LIN {X 0,Y 60.716,Z 312.384,A -85,B 0,C 180,E1 -29461.22,E2 -29461.22} C_VEL
LIN {X 0,Y 58.046,Z 307.358,A -85,B 0,C 180,E1 -29469.715,E2 -29469.715} C_VEL
LIN {X 0,Y 56.371,Z 305.582,A -85,B 0,C 180,E1 -29475.475,E2 -29475.475} C_VEL
LIN {X 0,Y 55.559,Z 303.266,A -85,B 0,C 180,E1 -29480.778,E2 -29480.778} C_VEL
LIN {X 0,Y 54.306,Z 302.152,A -85,B 0,C 180,E1 -29488.836,E2 -29488.836} C_VEL
LIN {X 0,Y 53.915,Z 301.998,A -85,B 0,C 180,E1 -29493.79,E2 -29493.79} C_VEL
LIN {X 0,Y 53.664,Z 302.515,A -85,B 0,C 180,E1 -29497.928,E2 -29497.928} C_VEL
LIN {X 0,Y 53.314,Z 303.941,A -85,B 0,C 180,E1 -29501.896,E2 -29501.896} C_VEL
LIN {X 0,Y 53.027,Z 308.841,A -85,B 0,C 180,E1 -29512.371,E2 -29512.371} C_VEL
LIN {X 0,Y 53.437,Z 309.628,A -85,B 0,C 180,E1 -29515.134,E2 -29515.134} C_VEL
LIN {X 0,Y 54.909,Z 313.062,A -85,B 0,C 180,E1 -29523.678,E2 -29523.678} C_VEL
LIN {X 0,Y 56.343,Z 316.547,A -85,B 0,C 180,E1 -29529.884,E2 -29529.884} C_VEL
LIN {X 0,Y 58.459,Z 322.301,A -85,B 0,C 180,E1 -29537.951,E2 -29537.951} C_VEL
LIN {X 0,Y 60.242,Z 328.035,A -85,B 0,C 180,E1 -29544.566,E2 -29544.566} C_VEL
LIN {X 0,Y 60.742,Z 331.305,A -85,B 0,C 180,E1 -29547.577,E2 -29547.577} C_VEL
LIN {X 0,Y 60.313,Z 334.364,A -85,B 0,C 180,E1 -29549.694,E2 -29549.694} C_VEL
LIN {X 0,Y 57.768,Z 345.368,A -85,B 0,C 180,E1 -29557.476,E2 -29557.476} C_VEL
LIN {X 0,Y 56.308,Z 350.331,A -85,B 0,C 180,E1 -29561.507,E2 -29561.507} C_VEL
LIN {X 0,Y 50.983,Z 359.168,A -85,B 0,C 180,E1 -29569.096,E2 -29569.096} C_VEL
LIN {X 0,Y 45.942,Z 367.817,A -85,B 0,C 180,E1 -29580.186,E2 -29580.186} C_VEL
LIN {X 0,Y 42.807,Z 374.789,A -85,B 0,C 180,E1 -29593.302,E2 -29593.302} C_VEL
LIN {X 0,Y 41.908,Z 379.494,A -85,B 0,C 180,E1 -29605.189,E2 -29605.189} C_VEL
LIN {X 0,Y 42.054,Z 382.623,A -85,B 0,C 180,E1 -29614.792,E2 -29614.792} C_VEL
LIN {X 0,Y 43.107,Z 386.22,A -85,B 0,C 180,E1 -29629.029,E2 -29629.029} C_VEL
LIN {X 0,Y 45.194,Z 388.132,A -85,B 0,C 180,E1 -29637.807,E2 -29637.807} C_VEL
LIN {X 0,Y 51.933,Z 390.826,A -85,B 0,C 180,E1 -29652.58,E2 -29652.58} C_VEL
LIN {X 0,Y 61.527,Z 392.195,A -85,B 0,C 180,E1 -29663.088,E2 -29663.088} C_VEL
LIN {X 0,Y 72.679,Z 392.248,A -85,B 0,C 180,E1 -29670.489,E2 -29670.489} C_VEL
LIN {X 0,Y 84.73,Z 390.994,A -85,B 0,C 180,E1 -29675.836,E2 -29675.836} C_VEL
LIN {X 0,Y 91.024,Z 389.845,A -85,B 0,C 180,E1 -29677.895,E2 -29677.895} C_VEL
LIN {X 0,Y 93.755,Z 389.205,A -85,B 0,C 180,E1 -29679.343,E2 -29679.343} C_VEL
LIN {X 0,Y 80.434,Z 391.186,A -85,B 0,C 180,E1 -29683.967,E2 -29683.967} C_VEL
LIN {X 0,Y 70.96,Z 391.617,A -85,B 0,C 180,E1 -29688.568,E2 -29688.568} C_VEL
LIN {X 0,Y 63.384,Z 391.312,A -85,B 0,C 180,E1 -29693.626,E2 -29693.626} C_VEL
LIN {X 0,Y 56.222,Z 390.333,A -85,B 0,C 180,E1 -29700.253,E2 -29700.253} C_VEL
LIN {X 0,Y 47.716,Z 387.672,A -85,B 0,C 180,E1 -29713.041,E2 -29713.041} C_VEL
LIN {X 0,Y 42.291,Z 383.509,A -85,B 0,C 180,E1 -29729.89,E2 -29729.89} C_VEL
LIN {X 0,Y 40.912,Z 378.594,A -85,B 0,C 180,E1 -29746.6,E2 -29746.6} C_VEL
LIN {X 0,Y 42.587,Z 372.224,A -85,B 0,C 180,E1 -29763.016,E2 -29763.016} C_VEL
LIN {X 0,Y 46.467,Z 364.513,A -85,B 0,C 180,E1 -29776.889,E2 -29776.889} C_VEL
LIN {X 0,Y 51.445,Z 356.174,A -85,B 0,C 180,E1 -29787.065,E2 -29787.065} C_VEL
LIN {X 0,Y 56.882,Z 347.135,A -85,B 0,C 180,E1 -29794.55,E2 -29794.55} C_VEL
LIN {X 0,Y 59.718,Z 342.179,A -85,B 0,C 180,E1 -29797.602,E2 -29797.602} C_VEL
LIN {X 0,Y 61.132,Z 334.574,A -85,B 0,C 180,E1 -29803.294,E2 -29803.294} C_VEL
LIN {X 0,Y 61.35,Z 332.923,A -85,B 0,C 180,E1 -29804.489,E2 -29804.489} C_VEL
LIN {X 0,Y 60.3,Z 328.115,A -85,B 0,C 180,E1 -29809.376,E2 -29809.376} C_VEL
LIN {X 0,Y 59.125,Z 324.115,A -85,B 0,C 180,E1 -29813.986,E2 -29813.986} C_VEL
LIN {X 0,Y 56.439,Z 317.616,A -85,B 0,C 180,E1 -29823.356,E2 -29823.356} C_VEL
LIN {X 0,Y 54.803,Z 314.262,A -85,B 0,C 180,E1 -29829.882,E2 -29829.882} C_VEL
LIN {X 0,Y 52.508,Z 309.531,A -85,B 0,C 180,E1 -29843.426,E2 -29843.426} C_VEL
LIN {X 0,Y 51.489,Z 308.683,A -85,B 0,C 180,E1 -29854.149,E2 -29854.149} C_VEL
LIN {X 0,Y 51.797,Z 308.515,A -85,B 0,C 180,E1 -29864.264,E2 -29864.264} C_VEL
LIN {X 0,Y 52.94,Z 309.058,A -85,B 0,C 180,E1 -29872.38,E2 -29872.38} C_VEL
LIN {X 0,Y 53.437,Z 309.628,A -85,B 0,C 180,E1 -29875.134,E2 -29875.134} C_VEL
LIN {X 0,Y 54.073,Z 310.974,A -85,B 0,C 180,E1 -29878.941,E2 -29878.941} C_VEL
LIN {X 0,Y 54.486,Z 314.348,A -85,B 0,C 180,E1 -29884.001,E2 -29884.001} C_VEL
LIN {X 0,Y 54.414,Z 318.577,A -85,B 0,C 180,E1 -29888.441,E2 -29888.441} C_VEL
LIN {X 0,Y 54.152,Z 327.952,A -85,B 0,C 180,E1 -29897.401,E2 -29897.401} C_VEL
LIN {X 0,Y 54.569,Z 330.721,A -85,B 0,C 180,E1 -29900.693,E2 -29900.693} C_VEL
LIN {X 0,Y 54.973,Z 334.381,A -85,B 0,C 180,E1 -29904.759,E2 -29904.759} C_VEL
LIN {X 0,Y 52.046,Z 344.757,A -85,B 0,C 180,E1 -29912.704,E2 -29912.704} C_VEL
LIN {X 0,Y 50.55,Z 349.485,A -85,B 0,C 180,E1 -29916.925,E2 -29916.925} C_VEL
LIN {X 0,Y 44.772,Z 358.482,A -85,B 0,C 180,E1 -29925.058,E2 -29925.058} C_VEL
LIN {X 0,Y 39.175,Z 367.209,A -85,B 0,C 180,E1 -29937.437,E2 -29937.437} C_VEL
LIN {X 0,Y 35.705,Z 374.24,A -85,B 0,C 180,E1 -29952.826,E2 -29952.826} C_VEL
LIN {X 0,Y 34.905,Z 379.848,A -85,B 0,C 180,E1 -29969.998,E2 -29969.998} C_VEL
LIN {X 0,Y 35.339,Z 382.791,A -85,B 0,C 180,E1 -29981.469,E2 -29981.469} C_VEL
LIN {X 0,Y 39.079,Z 387.199,A -85,B 0,C 180,E1 -30002.648,E2 -30002.648} C_VEL
LIN {X 0,Y 46.959,Z 390.173,A -85,B 0,C 180,E1 -30018.441,E2 -30018.441} C_VEL
LIN {X 0,Y 57.536,Z 391.813,A -85,B 0,C 180,E1 -30028.76,E2 -30028.76} C_VEL
LIN {X 0,Y 69.448,Z 392.107,A -85,B 0,C 180,E1 -30035.61,E2 -30035.61} C_VEL
LIN {X 0,Y 75.681,Z 391.763,A -85,B 0,C 180,E1 -30038.218,E2 -30038.218} C_VEL
LIN {X 0,Y 76.461,Z 391.653,A -85,B 0,C 180,E1 -30039.648,E2 -30039.648} C_VEL
LIN {X 0,Y 65.683,Z 391.772,A -85,B 0,C 180,E1 -30044.355,E2 -30044.355} C_VEL
LIN {X 0,Y 53.748,Z 390.589,A -85,B 0,C 180,E1 -30052.478,E2 -30052.478} C_VEL
LIN {X 0,Y 46.797,Z 389.001,A -85,B 0,C 180,E1 -30059.99,E2 -30059.99} C_VEL
LIN {X 0,Y 38.984,Z 385.698,A -85,B 0,C 180,E1 -30074.48,E2 -30074.48} C_VEL
LIN {X 0,Y 34.398,Z 380.739,A -85,B 0,C 180,E1 -30095.193,E2 -30095.193} C_VEL
LIN {X 0,Y 34.3,Z 375.093,A -85,B 0,C 180,E1 -30115.018,E2 -30115.018} C_VEL
LIN {X 0,Y 37.056,Z 368.741,A -85,B 0,C 180,E1 -30131.453,E2 -30131.453} C_VEL
LIN {X 0,Y 42.273,Z 360.323,A -85,B 0,C 180,E1 -30145.798,E2 -30145.798} C_VEL
LIN {X 0,Y 48.602,Z 350.774,A -85,B 0,C 180,E1 -30155.913,E2 -30155.913} C_VEL
LIN {X 0,Y 53.498,Z 343.032,A -85,B 0,C 180,E1 -30161.366,E2 -30161.366} C_VEL
LIN {X 0,Y 54.525,Z 339.734,A -85,B 0,C 180,E1 -30163.986,E2 -30163.986} C_VEL
LIN {X 0,Y 55.408,Z 334.818,A -85,B 0,C 180,E1 -30168.185,E2 -30168.185} C_VEL
LIN {X 0,Y 54.271,Z 329.443,A -85,B 0,C 180,E1 -30174.997,E2 -30174.997} C_VEL
LIN {X 0,Y 52.71,Z 324.789,A -85,B 0,C 180,E1 -30182.232,E2 -30182.232} C_VEL
LIN {X 0,Y 52.023,Z 322.703,A -85,B 0,C 180,E1 -30185.865,E2 -30185.865} C_VEL
LIN {X 0,Y 50.614,Z 319.24,A -85,B 0,C 180,E1 -30193.97,E2 -30193.97} C_VEL
LIN {X 0,Y 49.38,Z 315.79,A -85,B 0,C 180,E1 -30205.311,E2 -30205.311} C_VEL
LIN {X 0,Y 48.742,Z 315.216,A -85,B 0,C 180,E1 -30214.381,E2 -30214.381} C_VEL
LIN {X 0,Y 48.976,Z 315.067,A -85,B 0,C 180,E1 -30223.332,E2 -30223.332} C_VEL
LIN {X 0,Y 50.04,Z 315.547,A -85,B 0,C 180,E1 -30231.936,E2 -30231.936} C_VEL
LIN {X 0,Y 50.494,Z 316.572,A -85,B 0,C 180,E1 -30235.72,E2 -30235.72} C_VEL
LIN {X 0,Y 51.517,Z 319.997,A -85,B 0,C 180,E1 -30243.92,E2 -30243.92} C_VEL
LIN {X 0,Y 52.824,Z 324.176,A -85,B 0,C 180,E1 -30251.521,E2 -30251.521} C_VEL
LIN {X 0,Y 54.208,Z 329.381,A -85,B 0,C 180,E1 -30258.922,E2 -30258.922} C_VEL
LIN {X 0,Y 54.569,Z 330.721,A -85,B 0,C 180,E1 -30260.693,E2 -30260.693} C_VEL
LIN {X 0,Y 54.558,Z 332.559,A -85,B 0,C 180,E1 -30262.483,E2 -30262.483} C_VEL
LIN {X 0,Y 53.326,Z 335.803,A -85,B 0,C 180,E1 -30264.371,E2 -30264.371} C_VEL
LIN {X 0,Y 51.274,Z 339.05,A -85,B 0,C 180,E1 -30265.645,E2 -30265.645} C_VEL
LIN {X 0,Y 47.111,Z 344.69,A -85,B 0,C 180,E1 -30267.889,E2 -30267.889} C_VEL
LIN {X 0,Y 45.301,Z 347.952,A -85,B 0,C 180,E1 -30270.404,E2 -30270.404} C_VEL
LIN {X 0,Y 43.976,Z 350.677,A -85,B 0,C 180,E1 -30272.962,E2 -30272.962} C_VEL
LIN {X 0,Y 37.684,Z 359.374,A -85,B 0,C 180,E1 -30281.754,E2 -30281.754} C_VEL
LIN {X 0,Y 31.666,Z 367.857,A -85,B 0,C 180,E1 -30296.297,E2 -30296.297} C_VEL
LIN {X 0,Y 28.279,Z 374.686,A -85,B 0,C 180,E1 -30315.608,E2 -30315.608} C_VEL
LIN {X 0,Y 28.17,Z 380.088,A -85,B 0,C 180,E1 -30337.164,E2 -30337.164} C_VEL
LIN {X 0,Y 31.613,Z 385.2,A -85,B 0,C 180,E1 -30363.762,E2 -30363.762} C_VEL
LIN {X 0,Y 37.538,Z 388.017,A -85,B 0,C 180,E1 -30378.491,E2 -30378.491} C_VEL
LIN {X 0,Y 48.259,Z 390.554,A -85,B 0,C 180,E1 -30390.897,E2 -30390.897} C_VEL
LIN {X 0,Y 60.433,Z 391.783,A -85,B 0,C 180,E1 -30398.485,E2 -30398.485} C_VEL
LIN {X 0,Y 60.519,Z 391.753,A -85,B 0,C 180,E1 -30399.603,E2 -30399.603} C_VEL
LIN {X 0,Y 50.89,Z 390.609,A -85,B 0,C 180,E1 -30405.168,E2 -30405.168} C_VEL
LIN {X 0,Y 42.516,Z 388.752,A -85,B 0,C 180,E1 -30412.648,E2 -30412.648} C_VEL
LIN {X 0,Y 33.366,Z 385.23,A -85,B 0,C 180,E1 -30427.617,E2 -30427.617} C_VEL
LIN {X 0,Y 27.735,Z 380.268,A -85,B 0,C 180,E1 -30450.431,E2 -30450.431} C_VEL
LIN {X 0,Y 27.244,Z 374.435,A -85,B 0,C 180,E1 -30475.377,E2 -30475.377} C_VEL
LIN {X 0,Y 30.793,Z 367.38,A -85,B 0,C 180,E1 -30496.809,E2 -30496.809} C_VEL
LIN {X 0,Y 35.668,Z 360.447,A -85,B 0,C 180,E1 -30510.002,E2 -30510.002} C_VEL
LIN {X 0,Y 41.664,Z 352.31,A -85,B 0,C 180,E1 -30519.712,E2 -30519.712} C_VEL
LIN {X 0,Y 48.311,Z 342.597,A -85,B 0,C 180,E1 -30526.916,E2 -30526.916} C_VEL
LIN {X 0,Y 49.59,Z 337.634,A -85,B 0,C 180,E1 -30531.654,E2 -30531.654} C_VEL
LIN {X 0,Y 48.943,Z 333.355,A -85,B 0,C 180,E1 -30537.942,E2 -30537.942} C_VEL
LIN {X 0,Y 47.869,Z 328.994,A -85,B 0,C 180,E1 -30545.964,E2 -30545.964} C_VEL
LIN {X 0,Y 46.91,Z 325.511,A -85,B 0,C 180,E1 -30554.351,E2 -30554.351} C_VEL
LIN {X 0,Y 46.141,Z 323.114,A -85,B 0,C 180,E1 -30562.477,E2 -30562.477} C_VEL
LIN {X 0,Y 45.657,Z 321.682,A -85,B 0,C 180,E1 -30572.509,E2 -30572.509} C_VEL
LIN {X 0,Y 45.787,Z 321.464,A -85,B 0,C 180,E1 -30582.133,E2 -30582.133} C_VEL
LIN {X 0,Y 46.731,Z 321.903,A -85,B 0,C 180,E1 -30591.361,E2 -30591.361} C_VEL
LIN {X 0,Y 47.022,Z 323.048,A -85,B 0,C 180,E1 -30595.404,E2 -30595.404} C_VEL
LIN {X 0,Y 47.743,Z 326.68,A -85,B 0,C 180,E1 -30604.231,E2 -30604.231} C_VEL
LIN {X 0,Y 48.495,Z 330.562,A -85,B 0,C 180,E1 -30611.504,E2 -30611.504} C_VEL
LIN {X 0,Y 49.287,Z 335.135,A -85,B 0,C 180,E1 -30618.591,E2 -30618.591} C_VEL
LIN {X 0,Y 49.339,Z 336.759,A -85,B 0,C 180,E1 -30620.603,E2 -30620.603} C_VEL
LIN {X 0,Y 45.669,Z 346.976,A -85,B 0,C 180,E1 -30629.433,E2 -30629.433} C_VEL
LIN {X 0,Y 45.301,Z 347.952,A -85,B 0,C 180,E1 -30630.404,E2 -30630.404} C_VEL
LIN {X 0,Y 43.757,Z 350.87,A -85,B 0,C 180,E1 -30633.014,E2 -30633.014} C_VEL
LIN {X 0,Y 41.514,Z 353.649,A -85,B 0,C 180,E1 -30635.127,E2 -30635.127} C_VEL
LIN {X 0,Y 38.792,Z 356.232,A -85,B 0,C 180,E1 -30636.972,E2 -30636.972} C_VEL
LIN {X 0,Y 28.057,Z 364.422,A -85,B 0,C 180,E1 -30645.277,E2 -30645.277} C_VEL
LIN {X 0,Y 24.543,Z 367.912,A -85,B 0,C 180,E1 -30653.085,E2 -30653.085} C_VEL
LIN {X 0,Y 20.966,Z 375.052,A -85,B 0,C 180,E1 -30680.349,E2 -30680.349} C_VEL
LIN {X 0,Y 21.261,Z 378.672,A -85,B 0,C 180,E1 -30699.51,E2 -30699.51} C_VEL
LIN {X 0,Y 22.751,Z 381.611,A -85,B 0,C 180,E1 -30717.601,E2 -30717.601} C_VEL
LIN {X 0,Y 28.253,Z 385.172,A -85,B 0,C 180,E1 -30738.262,E2 -30738.262} C_VEL
LIN {X 0,Y 39.035,Z 388.662,A -85,B 0,C 180,E1 -30754.179,E2 -30754.179} C_VEL
LIN {X 0,Y 45.234,Z 389.927,A -85,B 0,C 180,E1 -30758.776,E2 -30758.776} C_VEL
LIN {X 0,Y 45.057,Z 389.877,A -85,B 0,C 180,E1 -30759.364,E2 -30759.364} C_VEL
LIN {X 0,Y 34.775,Z 387.17,A -85,B 0,C 180,E1 -30768.326,E2 -30768.326} C_VEL
LIN {X 0,Y 24.541,Z 382.499,A -85,B 0,C 180,E1 -30787.983,E2 -30787.983} C_VEL
LIN {X 0,Y 20.01,Z 377.129,A -85,B 0,C 180,E1 -30817.832,E2 -30817.832} C_VEL
LIN {X 0,Y 21.004,Z 371.715,A -85,B 0,C 180,E1 -30845.323,E2 -30845.323} C_VEL
LIN {X 0,Y 25.297,Z 365.423,A -85,B 0,C 180,E1 -30866.02,E2 -30866.02} C_VEL
LIN {X 0,Y 31.266,Z 358.122,A -85,B 0,C 180,E1 -30879.707,E2 -30879.707} C_VEL
LIN {X 0,Y 39.257,Z 348.201,A -85,B 0,C 180,E1 -30889.726,E2 -30889.726} C_VEL
LIN {X 0,Y 43.096,Z 342.821,A -85,B 0,C 180,E1 -30893.252,E2 -30893.252} C_VEL
LIN {X 0,Y 43.721,Z 341.086,A -85,B 0,C 180,E1 -30895.02,E2 -30895.02} C_VEL
LIN {X 0,Y 43.82,Z 338.697,A -85,B 0,C 180,E1 -30898.762,E2 -30898.762} C_VEL
LIN {X 0,Y 43.376,Z 335.116,A -85,B 0,C 180,E1 -30905.911,E2 -30905.911} C_VEL
LIN {X 0,Y 43.101,Z 333.047,A -85,B 0,C 180,E1 -30910.711,E2 -30910.711} C_VEL
LIN {X 0,Y 42.589,Z 330.414,A -85,B 0,C 180,E1 -30918.71,E2 -30918.71} C_VEL
LIN {X 0,Y 42.234,Z 328.761,A -85,B 0,C 180,E1 -30926.309,E2 -30926.309} C_VEL
LIN {X 0,Y 42.137,Z 328.272,A -85,B 0,C 180,E1 -30929.989,E2 -30929.989} C_VEL
LIN {X 0,Y 42.261,Z 327.696,A -85,B 0,C 180,E1 -30940.585,E2 -30940.585} C_VEL
LIN {X 0,Y 43.067,Z 328.096,A -85,B 0,C 180,E1 -30950.619,E2 -30950.619} C_VEL
LIN {X 0,Y 43.323,Z 331.287,A -85,B 0,C 180,E1 -30960.011,E2 -30960.011} C_VEL
LIN {X 0,Y 43.54,Z 334.374,A -85,B 0,C 180,E1 -30966.964,E2 -30966.964} C_VEL
LIN {X 0,Y 43.802,Z 339.224,A -85,B 0,C 180,E1 -30975.697,E2 -30975.697} C_VEL
LIN {X 0,Y 39.58,Z 348.685,A -85,B 0,C 180,E1 -30984.752,E2 -30984.752} C_VEL
LIN {X 0,Y 39.077,Z 349.777,A -85,B 0,C 180,E1 -30985.939,E2 -30985.939} C_VEL
LIN {X 0,Y 32.076,Z 358.552,A -85,B 0,C 180,E1 -30994.749,E2 -30994.749} C_VEL
LIN {X 0,Y 25.114,Z 367.127,A -85,B 0,C 180,E1 -31010.973,E2 -31010.973} C_VEL
LIN {X 0,Y 24.543,Z 367.912,A -85,B 0,C 180,E1 -31013.085,E2 -31013.085} C_VEL
LIN {X 0,Y 21.759,Z 371.151,A -85,B 0,C 180,E1 -31023.248,E2 -31023.248} C_VEL
LIN {X 0,Y 18.795,Z 373.914,A -85,B 0,C 180,E1 -31035.659,E2 -31035.659} C_VEL
LIN {X 0,Y 16.594,Z 379.926,A -85,B 0,C 180,E1 -31085.347,E2 -31085.347} C_VEL
LIN {X 0,Y 18.464,Z 381.331,A -85,B 0,C 180,E1 -31096.13,E2 -31096.13} C_VEL
LIN {X 0,Y 24.149,Z 384.067,A -85,B 0,C 180,E1 -31110.811,E2 -31110.811} C_VEL
LIN {X 0,Y 28.293,Z 385.486,A -85,B 0,C 180,E1 -31120.58,E2 -31120.58} C_VEL
LIN {X 0,Y 17.858,Z 380.682,A -85,B 0,C 180,E1 -31139.973,E2 -31139.973} C_VEL
LIN {X 0,Y 13.183,Z 376.126,A -85,B 0,C 180,E1 -31172.173,E2 -31172.173} C_VEL
LIN {X 0,Y 14.585,Z 370.316,A -85,B 0,C 180,E1 -31214.399,E2 -31214.399} C_VEL
LIN {X 0,Y 21.494,Z 362.612,A -85,B 0,C 180,E1 -31241.32,E2 -31241.32} C_VEL
LIN {X 0,Y 29.787,Z 353.791,A -85,B 0,C 180,E1 -31253.836,E2 -31253.836} C_VEL
LIN {X 0,Y 38.015,Z 343.892,A -85,B 0,C 180,E1 -31260.559,E2 -31260.559} C_VEL
LIN {X 0,Y 38.475,Z 342.169,A -85,B 0,C 180,E1 -31263.23,E2 -31263.23} C_VEL
LIN {X 0,Y 38.462,Z 338.194,A -85,B 0,C 180,E1 -31273.056,E2 -31273.056} C_VEL
LIN {X 0,Y 38.311,Z 335.641,A -85,B 0,C 180,E1 -31282.301,E2 -31282.301} C_VEL
LIN {X 0,Y 38.287,Z 334.838,A -85,B 0,C 180,E1 -31286.601,E2 -31286.601} C_VEL
LIN {X 0,Y 38.371,Z 333.867,A -85,B 0,C 180,E1 -31298.525,E2 -31298.525} C_VEL
LIN {X 0,Y 39.057,Z 334.137,A -85,B 0,C 180,E1 -31309.646,E2 -31309.646} C_VEL
LIN {X 0,Y 38.819,Z 337.528,A -85,B 0,C 180,E1 -31320.012,E2 -31320.012} C_VEL
LIN {X 0,Y 38.564,Z 341.595,A -85,B 0,C 180,E1 -31329.188,E2 -31329.188} C_VEL
LIN {X 0,Y 34.138,Z 349.782,A -85,B 0,C 180,E1 -31337.793,E2 -31337.793} C_VEL
LIN {X 0,Y 25.651,Z 359.282,A -85,B 0,C 180,E1 -31347.069,E2 -31347.069} C_VEL
LIN {X 0,Y 17.786,Z 367.686,A -85,B 0,C 180,E1 -31366.247,E2 -31366.247} C_VEL
LIN {X 0,Y 14.111,Z 373.368,A -85,B 0,C 180,E1 -31395.576,E2 -31395.576} C_VEL
LIN {X 0,Y 14.415,Z 377.198,A -85,B 0,C 180,E1 -31424.105,E2 -31424.105} C_VEL
LIN {X 0,Y 18.464,Z 381.331,A -85,B 0,C 180,E1 -31456.13,E2 -31456.13} C_VEL
LIN {X 0,Y 18.545,Z 381.531,A -85,B 0,C 180,E1 -31459.715,E2 -31459.715} C_VEL
LIN {X 0,Y 17.357,Z 381.21,A -85,B 0,C 180,E1 -31465.96,E2 -31465.96} C_VEL
LIN {X 0,Y 14.313,Z 379.893,A -85,B 0,C 180,E1 -31475.435,E2 -31475.435} C_VEL
LIN {X 0,Y 8.464,Z 376.55,A -85,B 0,C 180,E1 -31497.879,E2 -31497.879} C_VEL
LIN {X 0,Y 5.872,Z 372.951,A -85,B 0,C 180,E1 -31548.256,E2 -31548.256} C_VEL
LIN {X 0,Y 11.855,Z 366.333,A -85,B 0,C 180,E1 -31607.265,E2 -31607.265} C_VEL
LIN {X 0,Y 20.17,Z 359.068,A -85,B 0,C 180,E1 -31621.514,E2 -31621.514} C_VEL
LIN {X 0,Y 29.738,Z 349.384,A -85,B 0,C 180,E1 -31628.345,E2 -31628.345} C_VEL
LIN {X 0,Y 32.922,Z 345.7,A -85,B 0,C 180,E1 -31629.825,E2 -31629.825} C_VEL
LIN {X 0,Y 33.51,Z 344.116,A -85,B 0,C 180,E1 -31633.186,E2 -31633.186} C_VEL
LIN {X 0,Y 33.842,Z 341.722,A -85,B 0,C 180,E1 -31641.482,E2 -31641.482} C_VEL
LIN {X 0,Y 33.966,Z 340.854,A -85,B 0,C 180,E1 -31645.861,E2 -31645.861} C_VEL
LIN {X 0,Y 34.166,Z 339.904,A -85,B 0,C 180,E1 -31655.723,E2 -31655.723} C_VEL
LIN {X 0,Y 34.696,Z 340.019,A -85,B 0,C 180,E1 -31668.327,E2 -31668.327} C_VEL
LIN {X 0,Y 34.037,Z 342.627,A -85,B 0,C 180,E1 -31677.055,E2 -31677.055} C_VEL
LIN {X 0,Y 33.678,Z 344.323,A -85,B 0,C 180,E1 -31681.509,E2 -31681.509} C_VEL
LIN {X 0,Y 30.038,Z 349.829,A -85,B 0,C 180,E1 -31687.26,E2 -31687.26} C_VEL
LIN {X 0,Y 19.987,Z 359.933,A -85,B 0,C 180,E1 -31694.753,E2 -31694.753} C_VEL
LIN {X 0,Y 10.762,Z 368.118,A -85,B 0,C 180,E1 -31715.275,E2 -31715.275} C_VEL
LIN {X 0,Y 6.917,Z 373.66,A -85,B 0,C 180,E1 -31769.991,E2 -31769.991} C_VEL
LIN {X 0,Y 7.864,Z 375.572,A -85,B 0,C 180,E1 -31796.531,E2 -31796.531} C_VEL
LIN {X 0,Y 11.266,Z 378.267,A -85,B 0,C 180,E1 -31825.133,E2 -31825.133} C_VEL
LIN {X 0,Y 13.778,Z 379.611,A -85,B 0,C 180,E1 -31839.108,E2 -31839.108} C_VEL
LIN {X 0,Y 6.406,Z 374.605,A -85,B 0,C 180,E1 -31881.397,E2 -31881.397} C_VEL
LIN {X 0,Y 5.872,Z 372.951,A -85,B 0,C 180,E1 -31908.256,E2 -31908.256} C_VEL
LIN {X 0,Y 7.311,Z 369.812,A -85,B 0,C 180,E1 -31950.794,E2 -31950.794} C_VEL
LIN {X 0,Y 10.251,Z 366.357,A -85,B 0,C 180,E1 -31976.271,E2 -31976.271} C_VEL
LIN {X 0,Y 19.301,Z 357.358,A -85,B 0,C 180,E1 -32000.081,E2 -32000.081} C_VEL
LIN {X 0,Y 23.585,Z 353.135,A -85,B 0,C 180,E1 -32001.864,E2 -32001.864} C_VEL
LIN {X 0,Y 28.914,Z 347.476,A -85,B 0,C 180,E1 -32002.024,E2 -32002.024} C_VEL
LIN {X 0,Y 29.49,Z 345.902,A -85,B 0,C 180,E1 -32011.553,E2 -32011.553} C_VEL
LIN {X 0,Y 29.779,Z 345.508,A -85,B 0,C 180,E1 -32020.744,E2 -32020.744} C_VEL
LIN {X 0,Y 29.966,Z 345.678,A -85,B 0,C 180,E1 -32026.453,E2 -32026.453} C_VEL
LIN {X 0,Y 29.581,Z 346.507,A -85,B 0,C 180,E1 -32029.767,E2 -32029.767} C_VEL
LIN {X 0,Y 28.328,Z 348.4,A -85,B 0,C 180,E1 -32032.921,E2 -32032.921} C_VEL
LIN {X 0,Y 27.248,Z 349.716,A -85,B 0,C 180,E1 -32033.96,E2 -32033.96} C_VEL
LIN {X 0,Y 17.654,Z 358.962,A -85,B 0,C 180,E1 -32034.429,E2 -32034.429} C_VEL
LIN {X 0,Y 7.056,Z 367.277,A -85,B 0,C 180,E1 -32034.971,E2 -32034.971} C_VEL
LIN {X 0,Y 5.814,Z 368.137,A -85,B 0,C 180,E1 -32034.781,E2 -32034.781} C_VEL
LIN {X 0,Y 3.678,Z 369.417,A -85,B 0,C 180,E1 -32012.602,E2 -32012.602} C_VEL
LIN {X 0,Y 13.443,Z 362.235,A -85,B 0,C 180,E1 -32002.268,E2 -32002.268} C_VEL
LIN {X 0,Y 23.585,Z 353.135,A -85,B 0,C 180,E1 -32001.864,E2 -32001.864} C_VEL
LIN {X 0,Y 26.971,Z 354.577,A -85,B 0,C 180,E1 -32001.769,E2 -32001.769} C_VEL
LIN {X 0,Y 26.971,Z 600,A -85,B 0,C 180,E1 -32001.769,E2 -32001.769} C_VEL
LIN {X 0,Y 26.971,Z 600,A -85,B 0,C 180,E1 -32001.769,E2 -32001.769}

QRS_NEXT_CUT()

QRS_NEXT()
QRS_HOME()

END
